LIN {X 0,Y 300.85,Z 546.983,A -85,B 0,C 180,E1 1983.68,E2 1983.68} C_VEL
LIN {X 0,Y 306.335,Z 523.084,A -85,B 0,C 180,E1 1983.212,E2 1983.212} C_VEL
LIN {X 0,Y 309.917,Z 499.874,A -85,B 0,C 180,E1 1982.824,E2 1982.824} C_VEL
LIN {X 0,Y 321.366,Z 402.053,A -85,B 0,C 180,E1 1981.248,E2 1981.248} C_VEL
LIN {X 0,Y 320.937,Z 400.568,A -85,B 0,C 180,E1 1978.393,E2 1978.393} C_VEL
LIN {X 0,Y 321.124,Z 402.876,A -85,B 0,C 180,E1 1974.448,E2 1974.448} C_VEL
LIN {X 0,Y 307.919,Z 513.947,A -85,B 0,C 180,E1 1972.759,E2 1972.759} C_VEL
LIN {X 0,Y 303.476,Z 536.476,A -85,B 0,C 180,E1 1972.375,E2 1972.375} C_VEL
LIN {X 0,Y 297.372,Z 559.018,A -85,B 0,C 180,E1 1971.893,E2 1971.893} C_VEL
LIN {X 0,Y 290.292,Z 579.356,A -85,B 0,C 180,E1 1971.299,E2 1971.299} C_VEL
LIN {X 0,Y 281.315,Z 600.354,A -85,B 0,C 180,E1 1970.495,E2 1970.495} C_VEL
LIN {X 0,Y 271.469,Z 619.823,A -85,B 0,C 180,E1 1969.536,E2 1969.536} C_VEL
LIN {X 0,Y 260.309,Z 638.411,A -85,B 0,C 180,E1 1968.361,E2 1968.361} C_VEL
LIN {X 0,Y 247.458,Z 657.08,A -85,B 0,C 180,E1 1966.84,E2 1966.84} C_VEL
LIN {X 0,Y 234.799,Z 673.136,A -85,B 0,C 180,E1 1965.155,E2 1965.155} C_VEL
LIN {X 0,Y 220.615,Z 688.99,A -85,B 0,C 180,E1 1962.99,E2 1962.99} C_VEL
LIN {X 0,Y 205.942,Z 703.636,A -85,B 0,C 180,E1 1960.365,E2 1960.365} C_VEL
LIN {X 0,Y 190.94,Z 716.802,A -85,B 0,C 180,E1 1957.161,E2 1957.161} C_VEL
LIN {X 0,Y 175.091,Z 729.345,A -85,B 0,C 180,E1 1952.976,E2 1952.976} C_VEL
LIN {X 0,Y 160.324,Z 739.898,A -85,B 0,C 180,E1 1948.01,E2 1948.01} C_VEL
LIN {X 0,Y 146.292,Z 748.96,A -85,B 0,C 180,E1 1941.81,E2 1941.81} C_VEL
LIN {X 0,Y 133.673,Z 756.634,A -85,B 0,C 180,E1 1934.076,E2 1934.076} C_VEL
LIN {X 0,Y 123.681,Z 762.5,A -85,B 0,C 180,E1 1925.027,E2 1925.027} C_VEL
LIN {X 0,Y 116.775,Z 766.633,A -85,B 0,C 180,E1 1914.805,E2 1914.805} C_VEL
LIN {X 0,Y 113.23,Z 769.201,A -85,B 0,C 180,E1 1904.314,E2 1904.314} C_VEL
LIN {X 0,Y 112.174,Z 770.206,A -85,B 0,C 180,E1 1894.601,E2 1894.601} C_VEL
LIN {X 0,Y 112.127,Z 770.283,A -85,B 0,C 180,E1 1887.118,E2 1887.118} C_VEL
LIN {X 0,Y 112.706,Z 769.615,A -85,B 0,C 180,E1 1878.746,E2 1878.746} C_VEL
LIN {X 0,Y 115.591,Z 767.48,A -85,B 0,C 180,E1 1867.753,E2 1867.753} C_VEL
LIN {X 0,Y 121.421,Z 763.846,A -85,B 0,C 180,E1 1857.64,E2 1857.64} C_VEL
LIN {X 0,Y 131.081,Z 758.196,A -85,B 0,C 180,E1 1847.838,E2 1847.838} C_VEL
LIN {X 0,Y 143.143,Z 751.061,A -85,B 0,C 180,E1 1839.796,E2 1839.796} C_VEL
LIN {X 0,Y 157.037,Z 742.16,A -85,B 0,C 180,E1 1833.201,E2 1833.201} C_VEL
LIN {X 0,Y 171.955,Z 731.773,A -85,B 0,C 180,E1 1827.895,E2 1827.895} C_VEL
LIN {X 0,Y 186.811,Z 720.428,A -85,B 0,C 180,E1 1823.765,E2 1823.765} C_VEL
LIN {X 0,Y 201.625,Z 707.683,A -85,B 0,C 180,E1 1820.41,E2 1820.41} C_VEL
LIN {X 0,Y 217.043,Z 692.931,A -85,B 0,C 180,E1 1817.529,E2 1817.529} C_VEL
LIN {X 0,Y 231.146,Z 677.659,A -85,B 0,C 180,E1 1815.292,E2 1815.292} C_VEL
LIN {X 0,Y 245.108,Z 660.462,A -85,B 0,C 180,E1 1813.375,E2 1813.375} C_VEL
LIN {X 0,Y 257.937,Z 642.496,A -85,B 0,C 180,E1 1811.832,E2 1811.832} C_VEL
LIN {X 0,Y 269.068,Z 624.347,A -85,B 0,C 180,E1 1810.625,E2 1810.625} C_VEL
LIN {X 0,Y 280.314,Z 602.942,A -85,B 0,C 180,E1 1809.521,E2 1809.521} C_VEL
LIN {X 0,Y 289.288,Z 582.628,A -85,B 0,C 180,E1 1808.711,E2 1808.711} C_VEL
LIN {X 0,Y 296.888,Z 561.22,A -85,B 0,C 180,E1 1808.067,E2 1808.067} C_VEL
LIN {X 0,Y 303.507,Z 537.366,A -85,B 0,C 180,E1 1807.547,E2 1807.547} C_VEL
LIN {X 0,Y 308.067,Z 514.578,A -85,B 0,C 180,E1 1807.157,E2 1807.157} C_VEL
LIN {X 0,Y 318.488,Z 427.457,A -85,B 0,C 180,E1 1805.83,E2 1805.83} C_VEL
LIN {X 0,Y 321.368,Z 402.948,A -85,B 0,C 180,E1 1805.445,E2 1805.445} C_VEL
LIN {X 0,Y 321.176,Z 400.924,A -85,B 0,C 180,E1 1801.427,E2 1801.427} C_VEL
LIN {X 0,Y 321.579,Z 402.546,A -85,B 0,C 180,E1 1798.708,E2 1798.708} C_VEL
LIN {X 0,Y 308.318,Z 513.24,A -85,B 0,C 180,E1 1796.963,E2 1796.963} C_VEL
LIN {X 0,Y 305.949,Z 526.418,A -85,B 0,C 180,E1 1796.734,E2 1796.734} C_VEL
LIN {X 0,Y 304.314,Z 534.011,A -85,B 0,C 180,E1 1796.782,E2 1796.782} C_VEL
LIN {X 0,Y 298.825,Z 552.994,A -85,B 0,C 180,E1 1797.537,E2 1797.537} C_VEL
LIN {X 0,Y 296.424,Z 560.346,A -85,B 0,C 180,E1 1797.555,E2 1797.555} C_VEL
LIN {X 0,Y 288.862,Z 581.554,A -85,B 0,C 180,E1 1796.943,E2 1796.943} C_VEL
LIN {X 0,Y 280.061,Z 601.523,A -85,B 0,C 180,E1 1796.2,E2 1796.2} C_VEL
LIN {X 0,Y 269.874,Z 621.266,A -85,B 0,C 180,E1 1795.268,E2 1795.268} C_VEL
LIN {X 0,Y 258.314,Z 640.207,A -85,B 0,C 180,E1 1794.122,E2 1794.122} C_VEL
LIN {X 0,Y 244.7,Z 659.572,A -85,B 0,C 180,E1 1792.608,E2 1792.608} C_VEL
LIN {X 0,Y 230.893,Z 676.781,A -85,B 0,C 180,E1 1790.86,E2 1790.86} C_VEL
LIN {X 0,Y 215.849,Z 693.137,A -85,B 0,C 180,E1 1788.663,E2 1788.663} C_VEL
LIN {X 0,Y 199.979,Z 708.528,A -85,B 0,C 180,E1 1785.915,E2 1785.915} C_VEL
LIN {X 0,Y 184.365,Z 722.031,A -85,B 0,C 180,E1 1782.644,E2 1782.644} C_VEL
LIN {X 0,Y 167.831,Z 734.817,A -85,B 0,C 180,E1 1778.333,E2 1778.333} C_VEL
LIN {X 0,Y 152.166,Z 745.889,A -85,B 0,C 180,E1 1773.039,E2 1773.039} C_VEL
LIN {X 0,Y 137.685,Z 755.245,A -85,B 0,C 180,E1 1766.503,E2 1766.503} C_VEL
LIN {X 0,Y 124.167,Z 763.536,A -85,B 0,C 180,E1 1757.8,E2 1757.8} C_VEL
LIN {X 0,Y 114.104,Z 769.775,A -85,B 0,C 180,E1 1747.834,E2 1747.834} C_VEL
LIN {X 0,Y 107.643,Z 774.053,A -85,B 0,C 180,E1 1736.913,E2 1736.913} C_VEL
LIN {X 0,Y 104.582,Z 776.871,A -85,B 0,C 180,E1 1725.527,E2 1725.527} C_VEL
LIN {X 0,Y 104.042,Z 778.016,A -85,B 0,C 180,E1 1715.515,E2 1715.515} C_VEL
LIN {X 0,Y 104.082,Z 778.19,A -85,B 0,C 180,E1 1708.349,E2 1708.349} C_VEL
LIN {X 0,Y 104.104,Z 777.613,A -85,B 0,C 180,E1 1700.045,E2 1700.045} C_VEL
LIN {X 0,Y 105.275,Z 776.015,A -85,B 0,C 180,E1 1690.585,E2 1690.585} C_VEL
LIN {X 0,Y 109.559,Z 772.724,A -85,B 0,C 180,E1 1679.076,E2 1679.076} C_VEL
LIN {X 0,Y 117.382,Z 767.616,A -85,B 0,C 180,E1 1668.365,E2 1668.365} C_VEL
LIN {X 0,Y 128.576,Z 760.822,A -85,B 0,C 180,E1 1658.957,E2 1658.957} C_VEL
LIN {X 0,Y 141.779,Z 752.578,A -85,B 0,C 180,E1 1651.428,E2 1651.428} C_VEL
LIN {X 0,Y 156.899,Z 742.51,A -85,B 0,C 180,E1 1645.192,E2 1645.192} C_VEL
LIN {X 0,Y 172.685,Z 731.153,A -85,B 0,C 180,E1 1640.288,E2 1640.288} C_VEL
LIN {X 0,Y 188.628,Z 718.295,A -85,B 0,C 180,E1 1636.383,E2 1636.383} C_VEL
LIN {X 0,Y 205.301,Z 703.363,A -85,B 0,C 180,E1 1633.09,E2 1633.09} C_VEL
LIN {X 0,Y 220.713,Z 687.911,A -85,B 0,C 180,E1 1630.577,E2 1630.577} C_VEL
LIN {X 0,Y 235.174,Z 671.347,A -85,B 0,C 180,E1 1628.557,E2 1628.557} C_VEL
LIN {X 0,Y 249.238,Z 653.14,A -85,B 0,C 180,E1 1626.852,E2 1626.852} C_VEL
LIN {X 0,Y 261.669,Z 634.646,A -85,B 0,C 180,E1 1625.518,E2 1625.518} C_VEL
LIN {X 0,Y 273.256,Z 614.539,A -85,B 0,C 180,E1 1624.393,E2 1624.393} C_VEL
LIN {X 0,Y 282.991,Z 594.865,A -85,B 0,C 180,E1 1623.536,E2 1623.536} C_VEL
LIN {X 0,Y 291.31,Z 574.448,A -85,B 0,C 180,E1 1622.845,E2 1622.845} C_VEL
LIN {X 0,Y 298.806,Z 551.771,A -85,B 0,C 180,E1 1622.256,E2 1622.256} C_VEL
LIN {X 0,Y 304.384,Z 529.797,A -85,B 0,C 180,E1 1621.828,E2 1621.828} C_VEL
LIN {X 0,Y 308.359,Z 506.904,A -85,B 0,C 180,E1 1621.453,E2 1621.453} C_VEL
LIN {X 0,Y 320.097,Z 409.255,A -85,B 0,C 180,E1 1619.96,E2 1619.96} C_VEL
LIN {X 0,Y 319.937,Z 408.589,A -85,B 0,C 180,E1 1618.209,E2 1618.209} C_VEL
LIN {X 0,Y 319.912,Z 410.101,A -85,B 0,C 180,E1 1615.774,E2 1615.774} C_VEL
LIN {X 0,Y 307.308,Z 513.987,A -85,B 0,C 180,E1 1614.248,E2 1614.248} C_VEL
LIN {X 0,Y 302.797,Z 536.523,A -85,B 0,C 180,E1 1613.885,E2 1613.885} C_VEL
LIN {X 0,Y 296.587,Z 559.159,A -85,B 0,C 180,E1 1613.433,E2 1613.433} C_VEL
LIN {X 0,Y 289.674,Z 578.813,A -85,B 0,C 180,E1 1612.897,E2 1612.897} C_VEL
LIN {X 0,Y 280.584,Z 599.936,A -85,B 0,C 180,E1 1612.147,E2 1612.147} C_VEL
LIN {X 0,Y 270.603,Z 619.466,A -85,B 0,C 180,E1 1611.252,E2 1611.252} C_VEL
LIN {X 0,Y 259.277,Z 638.131,A -85,B 0,C 180,E1 1610.151,E2 1610.151} C_VEL
LIN {X 0,Y 246.212,Z 656.875,A -85,B 0,C 180,E1 1608.723,E2 1608.723} C_VEL
LIN {X 0,Y 232.859,Z 673.513,A -85,B 0,C 180,E1 1607.077,E2 1607.077} C_VEL
LIN {X 0,Y 218.38,Z 689.339,A -85,B 0,C 180,E1 1605.025,E2 1605.025} C_VEL
LIN {X 0,Y 203.355,Z 703.968,A -85,B 0,C 180,E1 1602.522,E2 1602.522} C_VEL
LIN {X 0,Y 187.821,Z 717.21,A -85,B 0,C 180,E1 1599.43,E2 1599.43} C_VEL
LIN {X 0,Y 170.734,Z 730.213,A -85,B 0,C 180,E1 1595.188,E2 1595.188} C_VEL
LIN {X 0,Y 155.403,Z 740.705,A -85,B 0,C 180,E1 1590.292,E2 1590.292} C_VEL
LIN {X 0,Y 140.71,Z 749.653,A -85,B 0,C 180,E1 1584.1,E2 1584.1} C_VEL
LIN {X 0,Y 126.808,Z 757.516,A -85,B 0,C 180,E1 1575.848,E2 1575.848} C_VEL
LIN {X 0,Y 116.248,Z 763.28,A -85,B 0,C 180,E1 1566.403,E2 1566.403} C_VEL
LIN {X 0,Y 108.918,Z 767.232,A -85,B 0,C 180,E1 1555.559,E2 1555.559} C_VEL
LIN {X 0,Y 105.094,Z 769.696,A -85,B 0,C 180,E1 1543.759,E2 1543.759} C_VEL
LIN {X 0,Y 104.17,Z 770.517,A -85,B 0,C 180,E1 1534.404,E2 1534.404} C_VEL
LIN {X 0,Y 104.138,Z 770.566,A -85,B 0,C 180,E1 1526.698,E2 1526.698} C_VEL
LIN {X 0,Y 104.809,Z 769.907,A -85,B 0,C 180,E1 1517.885,E2 1517.885} C_VEL
LIN {X 0,Y 107.958,Z 767.878,A -85,B 0,C 180,E1 1506.478,E2 1506.478} C_VEL
LIN {X 0,Y 114.601,Z 764.142,A -85,B 0,C 180,E1 1495.452,E2 1495.452} C_VEL
LIN {X 0,Y 125.128,Z 758.495,A -85,B 0,C 180,E1 1485.319,E2 1485.319} C_VEL
LIN {X 0,Y 138.038,Z 751.362,A -85,B 0,C 180,E1 1477.18,E2 1477.18} C_VEL
LIN {X 0,Y 152.396,Z 742.65,A -85,B 0,C 180,E1 1470.744,E2 1470.744} C_VEL
LIN {X 0,Y 168.282,Z 732.081,A -85,B 0,C 180,E1 1465.433,E2 1465.433} C_VEL
LIN {X 0,Y 184.051,Z 720.452,A -85,B 0,C 180,E1 1461.345,E2 1461.345} C_VEL
LIN {X 0,Y 199.798,Z 707.246,A -85,B 0,C 180,E1 1458.048,E2 1458.048} C_VEL
LIN {X 0,Y 216.522,Z 691.447,A -85,B 0,C 180,E1 1455.182,E2 1455.182} C_VEL
LIN {X 0,Y 231.427,Z 675.489,A -85,B 0,C 180,E1 1453.037,E2 1453.037} C_VEL
LIN {X 0,Y 244.759,Z 659.044,A -85,B 0,C 180,E1 1451.365,E2 1451.365} C_VEL
LIN {X 0,Y 258.284,Z 640.025,A -85,B 0,C 180,E1 1449.876,E2 1449.876} C_VEL
LIN {X 0,Y 269.648,Z 621.523,A -85,B 0,C 180,E1 1448.758,E2 1448.758} C_VEL
LIN {X 0,Y 280.105,Z 601.418,A -85,B 0,C 180,E1 1447.816,E2 1447.816} C_VEL
LIN {X 0,Y 289.148,Z 580.835,A -85,B 0,C 180,E1 1447.068,E2 1447.068} C_VEL
LIN {X 0,Y 296.509,Z 560.122,A -85,B 0,C 180,E1 1446.495,E2 1446.495} C_VEL
LIN {X 0,Y 302.967,Z 536.836,A -85,B 0,C 180,E1 1446.027,E2 1446.027} C_VEL
LIN {X 0,Y 307.541,Z 514.047,A -85,B 0,C 180,E1 1445.66,E2 1445.66} C_VEL
LIN {X 0,Y 320.161,Z 410.157,A -85,B 0,C 180,E1 1444.13,E2 1444.13} C_VEL
LIN {X 0,Y 320.213,Z 408.924,A -85,B 0,C 180,E1 1441.253,E2 1441.253} C_VEL
LIN {X 0,Y 320.313,Z 409.713,A -85,B 0,C 180,E1 1440.029,E2 1440.029} C_VEL
LIN {X 0,Y 307.67,Z 513.462,A -85,B 0,C 180,E1 1438.447,E2 1438.447} C_VEL
LIN {X 0,Y 303.121,Z 536.211,A -85,B 0,C 180,E1 1438.064,E2 1438.064} C_VEL
LIN {X 0,Y 296.906,Z 558.879,A -85,B 0,C 180,E1 1437.591,E2 1437.591} C_VEL
LIN {X 0,Y 296.424,Z 560.346,A -85,B 0,C 180,E1 1437.555,E2 1437.555} C_VEL
LIN {X 0,Y 293.85,Z 567.982,A -85,B 0,C 180,E1 1437.556,E2 1437.556} C_VEL
LIN {X 0,Y 286.355,Z 586.249,A -85,B 0,C 180,E1 1438.198,E2 1438.198} C_VEL
LIN {X 0,Y 283.288,Z 593.171,A -85,B 0,C 180,E1 1438.161,E2 1438.161} C_VEL
LIN {X 0,Y 273.245,Z 613.523,A -85,B 0,C 180,E1 1437.351,E2 1437.351} C_VEL
LIN {X 0,Y 261.986,Z 633.058,A -85,B 0,C 180,E1 1436.353,E2 1436.353} C_VEL
LIN {X 0,Y 249.36,Z 651.677,A -85,B 0,C 180,E1 1435.125,E2 1435.125} C_VEL
LIN {X 0,Y 234.477,Z 670.763,A -85,B 0,C 180,E1 1433.48,E2 1433.48} C_VEL
LIN {X 0,Y 220.038,Z 687.044,A -85,B 0,C 180,E1 1431.639,E2 1431.639} C_VEL
LIN {X 0,Y 204.107,Z 702.714,A -85,B 0,C 180,E1 1429.272,E2 1429.272} C_VEL
LIN {X 0,Y 186.446,Z 718.124,A -85,B 0,C 180,E1 1426.078,E2 1426.078} C_VEL
LIN {X 0,Y 169.965,Z 730.956,A -85,B 0,C 180,E1 1422.359,E2 1422.359} C_VEL
LIN {X 0,Y 153.519,Z 742.298,A -85,B 0,C 180,E1 1417.64,E2 1417.64} C_VEL
LIN {X 0,Y 136.614,Z 752.921,A -85,B 0,C 180,E1 1411.116,E2 1411.116} C_VEL
LIN {X 0,Y 122.252,Z 761.316,A -85,B 0,C 180,E1 1403.272,E2 1403.272} C_VEL
LIN {X 0,Y 110.321,Z 767.897,A -85,B 0,C 180,E1 1393.528,E2 1393.528} C_VEL
LIN {X 0,Y 101.518,Z 773.023,A -85,B 0,C 180,E1 1381.466,E2 1381.466} C_VEL
LIN {X 0,Y 97.303,Z 775.984,A -85,B 0,C 180,E1 1369.821,E2 1369.821} C_VEL
LIN {X 0,Y 96.071,Z 777.613,A -85,B 0,C 180,E1 1358.378,E2 1358.378} C_VEL
LIN {X 0,Y 96.107,Z 777.966,A -85,B 0,C 180,E1 1350,E2 1350} C_VEL
LIN {X 0,Y 96.073,Z 777.583,A -85,B 0,C 180,E1 1341.368,E2 1341.368} C_VEL
LIN {X 0,Y 97.438,Z 775.84,A -85,B 0,C 180,E1 1329.581,E2 1329.581} C_VEL
LIN {X 0,Y 101.817,Z 772.822,A -85,B 0,C 180,E1 1317.976,E2 1317.976} C_VEL
LIN {X 0,Y 110.324,Z 767.845,A -85,B 0,C 180,E1 1306.468,E2 1306.468} C_VEL
LIN {X 0,Y 122.247,Z 761.249,A -85,B 0,C 180,E1 1296.725,E2 1296.725} C_VEL
LIN {X 0,Y 136.592,Z 752.85,A -85,B 0,C 180,E1 1288.889,E2 1288.889} C_VEL
LIN {X 0,Y 152.72,Z 742.723,A -85,B 0,C 180,E1 1282.617,E2 1282.617} C_VEL
LIN {X 0,Y 169.112,Z 731.441,A -85,B 0,C 180,E1 1277.849,E2 1277.849} C_VEL
LIN {X 0,Y 185.555,Z 718.683,A -85,B 0,C 180,E1 1274.094,E2 1274.094} C_VEL
LIN {X 0,Y 202.659,Z 703.879,A -85,B 0,C 180,E1 1270.955,E2 1270.955} C_VEL
LIN {X 0,Y 217.935,Z 688.97,A -85,B 0,C 180,E1 1268.637,E2 1268.637} C_VEL
LIN {X 0,Y 232.566,Z 672.763,A -85,B 0,C 180,E1 1266.736,E2 1266.736} C_VEL
LIN {X 0,Y 246.46,Z 655.418,A -85,B 0,C 180,E1 1265.169,E2 1265.169} C_VEL
LIN {X 0,Y 259.544,Z 636.425,A -85,B 0,C 180,E1 1263.858,E2 1263.858} C_VEL
LIN {X 0,Y 271.77,Z 615.824,A -85,B 0,C 180,E1 1262.762,E2 1262.762} C_VEL
LIN {X 0,Y 282.111,Z 595.339,A -85,B 0,C 180,E1 1261.922,E2 1261.922} C_VEL
LIN {X 0,Y 290.523,Z 574.999,A -85,B 0,C 180,E1 1261.28,E2 1261.28} C_VEL
LIN {X 0,Y 298.052,Z 552.671,A -85,B 0,C 180,E1 1260.736,E2 1260.736} C_VEL
LIN {X 0,Y 303.637,Z 531.077,A -85,B 0,C 180,E1 1260.34,E2 1260.34} C_VEL
LIN {X 0,Y 307.8,Z 507.983,A -85,B 0,C 180,E1 1259.98,E2 1259.98} C_VEL
LIN {X 0,Y 318.99,Z 416.494,A -85,B 0,C 180,E1 1258.608,E2 1258.608} C_VEL
LIN {X 0,Y 318.871,Z 417.333,A -85,B 0,C 180,E1 1257.109,E2 1257.109} C_VEL
LIN {X 0,Y 306.904,Z 514.026,A -85,B 0,C 180,E1 1255.742,E2 1255.742} C_VEL
LIN {X 0,Y 302.298,Z 536.708,A -85,B 0,C 180,E1 1255.398,E2 1255.398} C_VEL
LIN {X 0,Y 296.084,Z 559.1,A -85,B 0,C 180,E1 1254.983,E2 1254.983} C_VEL
LIN {X 0,Y 288.797,Z 579.545,A -85,B 0,C 180,E1 1254.466,E2 1254.466} C_VEL
LIN {X 0,Y 279.605,Z 600.515,A -85,B 0,C 180,E1 1253.769,E2 1253.769} C_VEL
LIN {X 0,Y 269.501,Z 619.982,A -85,B 0,C 180,E1 1252.935,E2 1252.935} C_VEL
LIN {X 0,Y 258.025,Z 638.579,A -85,B 0,C 180,E1 1251.91,E2 1251.91} C_VEL
LIN {X 0,Y 245.071,Z 656.875,A -85,B 0,C 180,E1 1250.607,E2 1250.607} C_VEL
LIN {X 0,Y 231.65,Z 673.342,A -85,B 0,C 180,E1 1249.087,E2 1249.087} C_VEL
LIN {X 0,Y 216.427,Z 689.686,A -85,B 0,C 180,E1 1247.099,E2 1247.099} C_VEL
LIN {X 0,Y 200.899,Z 704.438,A -85,B 0,C 180,E1 1244.705,E2 1244.705} C_VEL
LIN {X 0,Y 184.627,Z 717.92,A -85,B 0,C 180,E1 1241.693,E2 1241.693} C_VEL
LIN {X 0,Y 167.467,Z 730.525,A -85,B 0,C 180,E1 1237.728,E2 1237.728} C_VEL
LIN {X 0,Y 151.512,Z 741.011,A -85,B 0,C 180,E1 1232.983,E2 1232.983} C_VEL
LIN {X 0,Y 136.065,Z 749.956,A -85,B 0,C 180,E1 1226.897,E2 1226.897} C_VEL
LIN {X 0,Y 121.242,Z 757.813,A -85,B 0,C 180,E1 1218.628,E2 1218.628} C_VEL
LIN {X 0,Y 109.774,Z 763.578,A -85,B 0,C 180,E1 1208.936,E2 1208.936} C_VEL
LIN {X 0,Y 101.637,Z 767.528,A -85,B 0,C 180,E1 1197.539,E2 1197.539} C_VEL
LIN {X 0,Y 97.269,Z 769.99,A -85,B 0,C 180,E1 1184.891,E2 1184.891} C_VEL
LIN {X 0,Y 96.187,Z 770.808,A -85,B 0,C 180,E1 1174.77,E2 1174.77} C_VEL
LIN {X 0,Y 96.143,Z 770.868,A -85,B 0,C 180,E1 1166.748,E2 1166.748} C_VEL
LIN {X 0,Y 96.85,Z 770.262,A -85,B 0,C 180,E1 1157.479,E2 1157.479} C_VEL
LIN {X 0,Y 100.385,Z 768.276,A -85,B 0,C 180,E1 1145.012,E2 1145.012} C_VEL
LIN {X 0,Y 107.55,Z 764.636,A -85,B 0,C 180,E1 1133.489,E2 1133.489} C_VEL
LIN {X 0,Y 119.44,Z 758.793,A -85,B 0,C 180,E1 1122.554,E2 1122.554} C_VEL
LIN {X 0,Y 133.243,Z 751.663,A -85,B 0,C 180,E1 1114.369,E2 1114.369} C_VEL
LIN {X 0,Y 148.374,Z 742.949,A -85,B 0,C 180,E1 1108.024,E2 1108.024} C_VEL
LIN {X 0,Y 165.224,Z 732.188,A -85,B 0,C 180,E1 1102.787,E2 1102.787} C_VEL
LIN {X 0,Y 181.707,Z 720.409,A -85,B 0,C 180,E1 1098.841,E2 1098.841} C_VEL
LIN {X 0,Y 197.428,Z 707.566,A -85,B 0,C 180,E1 1095.802,E2 1095.802} C_VEL
LIN {X 0,Y 213.629,Z 692.698,A -85,B 0,C 180,E1 1093.224,E2 1093.224} C_VEL
LIN {X 0,Y 228.343,Z 677.36,A -85,B 0,C 180,E1 1091.242,E2 1091.242} C_VEL
LIN {X 0,Y 242.357,Z 660.631,A -85,B 0,C 180,E1 1089.605,E2 1089.605} C_VEL
LIN {X 0,Y 255.602,Z 642.645,A -85,B 0,C 180,E1 1088.25,E2 1088.25} C_VEL
LIN {X 0,Y 267.057,Z 624.485,A -85,B 0,C 180,E1 1087.194,E2 1087.194} C_VEL
LIN {X 0,Y 278.6,Z 603.078,A -85,B 0,C 180,E1 1086.233,E2 1086.233} C_VEL
LIN {X 0,Y 287.791,Z 582.774,A -85,B 0,C 180,E1 1085.531,E2 1085.531} C_VEL
LIN {X 0,Y 295.563,Z 561.409,A -85,B 0,C 180,E1 1084.973,E2 1084.973} C_VEL
LIN {X 0,Y 302.298,Z 537.76,A -85,B 0,C 180,E1 1084.526,E2 1084.526} C_VEL
LIN {X 0,Y 307.014,Z 514.966,A -85,B 0,C 180,E1 1084.18,E2 1084.18} C_VEL
LIN {X 0,Y 315.968,Z 443.369,A -85,B 0,C 180,E1 1083.167,E2 1083.167} C_VEL
LIN {X 0,Y 319.122,Z 417.372,A -85,B 0,C 180,E1 1082.784,E2 1082.784} C_VEL
LIN {X 0,Y 319.209,Z 416.958,A -85,B 0,C 180,E1 1081.36,E2 1081.36} C_VEL
LIN {X 0,Y 307.229,Z 513.683,A -85,B 0,C 180,E1 1079.937,E2 1079.937} C_VEL
LIN {X 0,Y 302.613,Z 536.45,A -85,B 0,C 180,E1 1079.576,E2 1079.576} C_VEL
LIN {X 0,Y 296.234,Z 559.362,A -85,B 0,C 180,E1 1079.129,E2 1079.129} C_VEL
LIN {X 0,Y 289.038,Z 579.526,A -85,B 0,C 180,E1 1078.596,E2 1078.596} C_VEL
LIN {X 0,Y 283.288,Z 593.171,A -85,B 0,C 180,E1 1078.161,E2 1078.161} C_VEL
LIN {X 0,Y 280.03,Z 600.219,A -85,B 0,C 180,E1 1078.108,E2 1078.108} C_VEL
LIN {X 0,Y 270.502,Z 617.76,A -85,B 0,C 180,E1 1078.649,E2 1078.649} C_VEL
LIN {X 0,Y 266.551,Z 624.394,A -85,B 0,C 180,E1 1078.554,E2 1078.554} C_VEL
LIN {X 0,Y 254.41,Z 643.457,A -85,B 0,C 180,E1 1077.523,E2 1077.523} C_VEL
LIN {X 0,Y 240.974,Z 661.506,A -85,B 0,C 180,E1 1076.254,E2 1076.254} C_VEL
LIN {X 0,Y 225.953,Z 679.199,A -85,B 0,C 180,E1 1074.63,E2 1074.63} C_VEL
LIN {X 0,Y 210.668,Z 694.954,A -85,B 0,C 180,E1 1072.709,E2 1072.709} C_VEL
LIN {X 0,Y 193.863,Z 710.172,A -85,B 0,C 180,E1 1070.201,E2 1070.201} C_VEL
LIN {X 0,Y 177.381,Z 723.486,A -85,B 0,C 180,E1 1067.196,E2 1067.196} C_VEL
LIN {X 0,Y 160.374,Z 735.563,A -85,B 0,C 180,E1 1063.335,E2 1063.335} C_VEL
LIN {X 0,Y 142.379,Z 747.005,A -85,B 0,C 180,E1 1057.964,E2 1057.964} C_VEL
LIN {X 0,Y 126.383,Z 756.231,A -85,B 0,C 180,E1 1051.418,E2 1051.418} C_VEL
LIN {X 0,Y 111.749,Z 763.877,A -85,B 0,C 180,E1 1042.778,E2 1042.778} C_VEL
LIN {X 0,Y 99.615,Z 770.049,A -85,B 0,C 180,E1 1031.486,E2 1031.486} C_VEL
LIN {X 0,Y 92.155,Z 774.09,A -85,B 0,C 180,E1 1019.224,E2 1019.224} C_VEL
LIN {X 0,Y 88.563,Z 776.584,A -85,B 0,C 180,E1 1005.721,E2 1005.721} C_VEL
LIN {X 0,Y 88.052,Z 777.458,A -85,B 0,C 180,E1 995.866,E2 995.866} C_VEL
LIN {X 0,Y 88.086,Z 777.608,A -85,B 0,C 180,E1 988.049,E2 988.049} C_VEL
LIN {X 0,Y 88.156,Z 777.098,A -85,B 0,C 180,E1 978.883,E2 978.883} C_VEL
LIN {X 0,Y 89.965,Z 775.418,A -85,B 0,C 180,E1 967.109,E2 967.109} C_VEL
LIN {X 0,Y 95.587,Z 772.178,A -85,B 0,C 180,E1 954.144,E2 954.144} C_VEL
LIN {X 0,Y 105.534,Z 766.979,A -85,B 0,C 180,E1 942.273,E2 942.273} C_VEL
LIN {X 0,Y 119.414,Z 759.837,A -85,B 0,C 180,E1 932.258,E2 932.258} C_VEL
LIN {X 0,Y 134.548,Z 751.54,A -85,B 0,C 180,E1 924.962,E2 924.962} C_VEL
LIN {X 0,Y 151.351,Z 741.345,A -85,B 0,C 180,E1 919.15,E2 919.15} C_VEL
LIN {X 0,Y 168.484,Z 729.852,A -85,B 0,C 180,E1 914.696,E2 914.696} C_VEL
LIN {X 0,Y 185.519,Z 716.924,A -85,B 0,C 180,E1 911.227,E2 911.227} C_VEL
LIN {X 0,Y 202.179,Z 702.674,A -85,B 0,C 180,E1 908.486,E2 908.486} C_VEL
LIN {X 0,Y 218.277,Z 687.196,A -85,B 0,C 180,E1 906.29,E2 906.29} C_VEL
LIN {X 0,Y 233.296,Z 670.57,A -85,B 0,C 180,E1 904.536,E2 904.536} C_VEL
LIN {X 0,Y 248.542,Z 651.277,A -85,B 0,C 180,E1 902.997,E2 902.997} C_VEL
LIN {X 0,Y 261.591,Z 632.222,A -85,B 0,C 180,E1 901.841,E2 901.841} C_VEL
LIN {X 0,Y 272.989,Z 612.554,A -85,B 0,C 180,E1 900.921,E2 900.921} C_VEL
LIN {X 0,Y 283.453,Z 591.256,A -85,B 0,C 180,E1 900.152,E2 900.152} C_VEL
LIN {X 0,Y 292.211,Z 569.689,A -85,B 0,C 180,E1 899.555,E2 899.555} C_VEL
LIN {X 0,Y 299.079,Z 548.087,A -85,B 0,C 180,E1 899.109,E2 899.109} C_VEL
LIN {X 0,Y 304.742,Z 524.632,A -85,B 0,C 180,E1 898.73,E2 898.73} C_VEL
LIN {X 0,Y 308.506,Z 501.749,A -85,B 0,C 180,E1 898.397,E2 898.397} C_VEL
LIN {X 0,Y 312.819,Z 466.535,A -85,B 0,C 180,E1 897.885,E2 897.885} C_VEL
LIN {X 0,Y 306.465,Z 515.586,A -85,B 0,C 180,E1 897.218,E2 897.218} C_VEL
LIN {X 0,Y 301.673,Z 538.312,A -85,B 0,C 180,E1 896.895,E2 896.895} C_VEL
LIN {X 0,Y 295.003,Z 561.412,A -85,B 0,C 180,E1 896.491,E2 896.491} C_VEL
LIN {X 0,Y 287.159,Z 582.778,A -85,B 0,C 180,E1 895.977,E2 895.977} C_VEL
LIN {X 0,Y 277.875,Z 603.085,A -85,B 0,C 180,E1 895.331,E2 895.331} C_VEL
LIN {X 0,Y 266.691,Z 623.692,A -85,B 0,C 180,E1 894.481,E2 894.481} C_VEL
LIN {X 0,Y 255.09,Z 641.932,A -85,B 0,C 180,E1 893.512,E2 893.512} C_VEL
LIN {X 0,Y 241.663,Z 660.068,A -85,B 0,C 180,E1 892.257,E2 892.257} C_VEL
LIN {X 0,Y 227.425,Z 676.917,A -85,B 0,C 180,E1 890.741,E2 890.741} C_VEL
LIN {X 0,Y 212.902,Z 691.858,A -85,B 0,C 180,E1 888.964,E2 888.964} C_VEL
LIN {X 0,Y 195.428,Z 707.66,A -85,B 0,C 180,E1 886.424,E2 886.424} C_VEL
LIN {X 0,Y 179.3,Z 720.519,A -85,B 0,C 180,E1 883.561,E2 883.561} C_VEL
LIN {X 0,Y 162.335,Z 732.297,A -85,B 0,C 180,E1 879.823,E2 879.823} C_VEL
LIN {X 0,Y 144.775,Z 743.107,A -85,B 0,C 180,E1 874.783,E2 874.783} C_VEL
LIN {X 0,Y 128.861,Z 751.835,A -85,B 0,C 180,E1 868.593,E2 868.593} C_VEL
LIN {X 0,Y 114.12,Z 758.99,A -85,B 0,C 180,E1 860.442,E2 860.442} C_VEL
LIN {X 0,Y 101.151,Z 764.862,A -85,B 0,C 180,E1 849.243,E2 849.243} C_VEL
LIN {X 0,Y 92.962,Z 768.595,A -85,B 0,C 180,E1 836.782,E2 836.782} C_VEL
LIN {X 0,Y 89.009,Z 770.532,A -85,B 0,C 180,E1 823.644,E2 823.644} C_VEL
LIN {X 0,Y 88.149,Z 771.161,A -85,B 0,C 180,E1 813.251,E2 813.251} C_VEL
LIN {X 0,Y 88.204,Z 771.107,A -85,B 0,C 180,E1 804.797,E2 804.797} C_VEL
LIN {X 0,Y 89.465,Z 770.307,A -85,B 0,C 180,E1 793.776,E2 793.776} C_VEL
LIN {X 0,Y 94.457,Z 767.878,A -85,B 0,C 180,E1 780.165,E2 780.165} C_VEL
LIN {X 0,Y 103.482,Z 763.945,A -85,B 0,C 180,E1 768.19,E2 768.19} C_VEL
LIN {X 0,Y 115.921,Z 758.214,A -85,B 0,C 180,E1 758.29,E2 758.29} C_VEL
LIN {X 0,Y 131.696,Z 750.392,A -85,B 0,C 180,E1 750.062,E2 750.062} C_VEL
LIN {X 0,Y 147.902,Z 741.457,A -85,B 0,C 180,E1 744.131,E2 744.131} C_VEL
LIN {X 0,Y 164.804,Z 730.792,A -85,B 0,C 180,E1 739.493,E2 739.493} C_VEL
LIN {X 0,Y 182.78,Z 717.975,A -85,B 0,C 180,E1 735.69,E2 735.69} C_VEL
LIN {X 0,Y 199.02,Z 704.853,A -85,B 0,C 180,E1 732.939,E2 732.939} C_VEL
LIN {X 0,Y 214.711,Z 690.298,A -85,B 0,C 180,E1 730.72,E2 730.72} C_VEL
LIN {X 0,Y 230.22,Z 674.027,A -85,B 0,C 180,E1 728.864,E2 728.864} C_VEL
LIN {X 0,Y 244.01,Z 657.41,A -85,B 0,C 180,E1 727.434,E2 727.434} C_VEL
LIN {X 0,Y 257.464,Z 638.72,A -85,B 0,C 180,E1 726.203,E2 726.203} C_VEL
LIN {X 0,Y 269.086,Z 620.122,A -85,B 0,C 180,E1 725.257,E2 725.257} C_VEL
LIN {X 0,Y 279.31,Z 600.657,A -85,B 0,C 180,E1 724.489,E2 724.489} C_VEL
LIN {X 0,Y 288.602,Z 579.719,A -85,B 0,C 180,E1 723.85,E2 723.85} C_VEL
LIN {X 0,Y 295.963,Z 559.299,A -85,B 0,C 180,E1 723.375,E2 723.375} C_VEL
LIN {X 0,Y 302.36,Z 536.489,A -85,B 0,C 180,E1 722.988,E2 722.988} C_VEL
LIN {X 0,Y 307.014,Z 513.722,A -85,B 0,C 180,E1 722.666,E2 722.666} C_VEL
LIN {X 0,Y 312.684,Z 469.731,A -85,B 0,C 180,E1 722.06,E2 722.06} C_VEL
LIN {X 0,Y 306.728,Z 515.57,A -85,B 0,C 180,E1 721.406,E2 721.406} C_VEL
LIN {X 0,Y 301.938,Z 538.268,A -85,B 0,C 180,E1 721.066,E2 721.066} C_VEL
LIN {X 0,Y 295.306,Z 561.246,A -85,B 0,C 180,E1 720.643,E2 720.643} C_VEL
LIN {X 0,Y 287.452,Z 582.663,A -85,B 0,C 180,E1 720.107,E2 720.107} C_VEL
LIN {X 0,Y 278.482,Z 602.35,A -85,B 0,C 180,E1 719.473,E2 719.473} C_VEL
LIN {X 0,Y 267.531,Z 622.769,A -85,B 0,C 180,E1 718.632,E2 718.632} C_VEL
LIN {X 0,Y 266.551,Z 624.394,A -85,B 0,C 180,E1 718.554,E2 718.554} C_VEL
LIN {X 0,Y 262.431,Z 631.157,A -85,B 0,C 180,E1 718.44,E2 718.44} C_VEL
LIN {X 0,Y 251.006,Z 647.521,A -85,B 0,C 180,E1 718.884,E2 718.884} C_VEL
LIN {X 0,Y 246.454,Z 653.632,A -85,B 0,C 180,E1 718.735,E2 718.735} C_VEL
LIN {X 0,Y 231.704,Z 671.703,A -85,B 0,C 180,E1 717.375,E2 717.375} C_VEL
LIN {X 0,Y 216.069,Z 688.483,A -85,B 0,C 180,E1 715.709,E2 715.709} C_VEL
LIN {X 0,Y 199.867,Z 703.661,A -85,B 0,C 180,E1 713.682,E2 713.682} C_VEL
LIN {X 0,Y 182.209,Z 718.188,A -85,B 0,C 180,E1 711.007,E2 711.007} C_VEL
LIN {X 0,Y 164.75,Z 730.931,A -85,B 0,C 180,E1 707.708,E2 707.708} C_VEL
LIN {X 0,Y 146.986,Z 742.264,A -85,B 0,C 180,E1 703.4,E2 703.4} C_VEL
LIN {X 0,Y 128.825,Z 752.578,A -85,B 0,C 180,E1 697.454,E2 697.454} C_VEL
LIN {X 0,Y 113.02,Z 760.704,A -85,B 0,C 180,E1 690.107,E2 690.107} C_VEL
LIN {X 0,Y 98.883,Z 767.289,A -85,B 0,C 180,E1 680.215,E2 680.215} C_VEL
LIN {X 0,Y 87.8,Z 772.423,A -85,B 0,C 180,E1 667.124,E2 667.124} C_VEL
LIN {X 0,Y 82.058,Z 775.389,A -85,B 0,C 180,E1 653.709,E2 653.709} C_VEL
LIN {X 0,Y 80.094,Z 777.048,A -85,B 0,C 180,E1 639.536,E2 639.536} C_VEL
LIN {X 0,Y 80.116,Z 777.384,A -85,B 0,C 180,E1 630,E2 630} C_VEL
LIN {X 0,Y 80.096,Z 777.043,A -85,B 0,C 180,E1 620.458,E2 620.458} C_VEL
LIN {X 0,Y 82.058,Z 775.365,A -85,B 0,C 180,E1 606.291,E2 606.291} C_VEL
LIN {X 0,Y 87.823,Z 772.38,A -85,B 0,C 180,E1 592.837,E2 592.837} C_VEL
LIN {X 0,Y 98.881,Z 767.236,A -85,B 0,C 180,E1 579.783,E2 579.783} C_VEL
LIN {X 0,Y 113.016,Z 760.63,A -85,B 0,C 180,E1 569.89,E2 569.89} C_VEL
LIN {X 0,Y 128.821,Z 752.487,A -85,B 0,C 180,E1 562.541,E2 562.541} C_VEL
LIN {X 0,Y 147.081,Z 742.09,A -85,B 0,C 180,E1 556.566,E2 556.566} C_VEL
LIN {X 0,Y 164.905,Z 730.7,A -85,B 0,C 180,E1 552.252,E2 552.252} C_VEL
LIN {X 0,Y 182.205,Z 718.029,A -85,B 0,C 180,E1 548.984,E2 548.984} C_VEL
LIN {X 0,Y 200.163,Z 703.193,A -85,B 0,C 180,E1 546.268,E2 546.268} C_VEL
LIN {X 0,Y 216.552,Z 687.792,A -85,B 0,C 180,E1 544.226,E2 544.226} C_VEL
LIN {X 0,Y 231.702,Z 671.433,A -85,B 0,C 180,E1 542.613,E2 542.613} C_VEL
LIN {X 0,Y 246.516,Z 653.209,A -85,B 0,C 180,E1 541.247,E2 541.247} C_VEL
LIN {X 0,Y 259.457,Z 634.769,A -85,B 0,C 180,E1 540.192,E2 540.192} C_VEL
LIN {X 0,Y 271.474,Z 614.751,A -85,B 0,C 180,E1 539.308,E2 539.308} C_VEL
LIN {X 0,Y 281.532,Z 595.167,A -85,B 0,C 180,E1 538.637,E2 538.637} C_VEL
LIN {X 0,Y 290.11,Z 574.799,A -85,B 0,C 180,E1 538.098,E2 538.098} C_VEL
LIN {X 0,Y 292.715,Z 567.909,A -85,B 0,C 180,E1 537.925,E2 537.925} C_VEL
LIN {X 0,Y 284.239,Z 589.029,A -85,B 0,C 180,E1 537.423,E2 537.423} C_VEL
LIN {X 0,Y 274.386,Z 609.457,A -85,B 0,C 180,E1 536.781,E2 536.781} C_VEL
LIN {X 0,Y 263.59,Z 628.189,A -85,B 0,C 180,E1 536.023,E2 536.023} C_VEL
LIN {X 0,Y 250.411,Z 647.789,A -85,B 0,C 180,E1 534.998,E2 534.998} C_VEL
LIN {X 0,Y 236.844,Z 665.272,A -85,B 0,C 180,E1 533.802,E2 533.802} C_VEL
LIN {X 0,Y 221.958,Z 681.783,A -85,B 0,C 180,E1 532.312,E2 532.312} C_VEL
LIN {X 0,Y 205.836,Z 697.496,A -85,B 0,C 180,E1 530.42,E2 530.42} C_VEL
LIN {X 0,Y 189.053,Z 711.776,A -85,B 0,C 180,E1 528.068,E2 528.068} C_VEL
LIN {X 0,Y 171.752,Z 724.596,A -85,B 0,C 180,E1 525.093,E2 525.093} C_VEL
LIN {X 0,Y 154.149,Z 736.101,A -85,B 0,C 180,E1 521.258,E2 521.258} C_VEL
LIN {X 0,Y 137.382,Z 745.649,A -85,B 0,C 180,E1 516.49,E2 516.49} C_VEL
LIN {X 0,Y 120.29,Z 754.221,A -85,B 0,C 180,E1 509.818,E2 509.818} C_VEL
LIN {X 0,Y 105.22,Z 761.009,A -85,B 0,C 180,E1 501.186,E2 501.186} C_VEL
LIN {X 0,Y 92.995,Z 765.948,A -85,B 0,C 180,E1 490.172,E2 490.172} C_VEL
LIN {X 0,Y 84.333,Z 769.422,A -85,B 0,C 180,E1 476.019,E2 476.019} C_VEL
LIN {X 0,Y 80.863,Z 771.013,A -85,B 0,C 180,E1 462.86,E2 462.86} C_VEL
LIN {X 0,Y 80.132,Z 771.516,A -85,B 0,C 180,E1 451.43,E2 451.43} C_VEL
LIN {X 0,Y 80.456,Z 771.301,A -85,B 0,C 180,E1 440.703,E2 440.703} C_VEL
LIN {X 0,Y 83.534,Z 769.78,A -85,B 0,C 180,E1 425.986,E2 425.986} C_VEL
LIN {X 0,Y 91.116,Z 766.801,A -85,B 0,C 180,E1 412.085,E2 412.085} C_VEL
LIN {X 0,Y 102.696,Z 762.067,A -85,B 0,C 180,E1 400.589,E2 400.589} C_VEL
LIN {X 0,Y 118.382,Z 755.198,A -85,B 0,C 180,E1 391.012,E2 391.012} C_VEL
LIN {X 0,Y 134.897,Z 747.127,A -85,B 0,C 180,E1 384.266,E2 384.266} C_VEL
LIN {X 0,Y 152.367,Z 737.256,A -85,B 0,C 180,E1 379.104,E2 379.104} C_VEL
LIN {X 0,Y 170.801,Z 725.399,A -85,B 0,C 180,E1 375.012,E2 375.012} C_VEL
LIN {X 0,Y 188.081,Z 712.759,A -85,B 0,C 180,E1 372.004,E2 372.004} C_VEL
LIN {X 0,Y 204.849,Z 698.569,A -85,B 0,C 180,E1 369.625,E2 369.625} C_VEL
LIN {X 0,Y 221.441,Z 682.566,A -85,B 0,C 180,E1 367.665,E2 367.665} C_VEL
LIN {X 0,Y 236.328,Z 666.179,A -85,B 0,C 180,E1 366.167,E2 366.167} C_VEL
LIN {X 0,Y 249.896,Z 648.827,A -85,B 0,C 180,E1 364.968,E2 364.968} C_VEL
LIN {X 0,Y 263.077,Z 629.445,A -85,B 0,C 180,E1 363.938,E2 363.938} C_VEL
LIN {X 0,Y 273.874,Z 610.839,A -85,B 0,C 180,E1 363.176,E2 363.176} C_VEL
LIN {X 0,Y 284.222,Z 589.641,A -85,B 0,C 180,E1 362.501,E2 362.501} C_VEL
LIN {X 0,Y 292.289,Z 569.856,A -85,B 0,C 180,E1 362.021,E2 362.021} C_VEL
LIN {X 0,Y 283.547,Z 591.172,A -85,B 0,C 180,E1 361.484,E2 361.484} C_VEL
LIN {X 0,Y 272.979,Z 612.474,A -85,B 0,C 180,E1 360.783,E2 360.783} C_VEL
LIN {X 0,Y 261.456,Z 632.143,A -85,B 0,C 180,E1 359.943,E2 359.943} C_VEL
LIN {X 0,Y 248.503,Z 650.839,A -85,B 0,C 180,E1 358.91,E2 358.91} C_VEL
LIN {X 0,Y 246.454,Z 653.632,A -85,B 0,C 180,E1 358.735,E2 358.735} C_VEL
LIN {X 0,Y 241.723,Z 659.756,A -85,B 0,C 180,E1 358.564,E2 358.564} C_VEL
LIN {X 0,Y 228.455,Z 674.839,A -85,B 0,C 180,E1 358.893,E2 358.893} C_VEL
LIN {X 0,Y 223.152,Z 680.407,A -85,B 0,C 180,E1 358.66,E2 358.66} C_VEL
LIN {X 0,Y 206.712,Z 696.634,A -85,B 0,C 180,E1 356.95,E2 356.95} C_VEL
LIN {X 0,Y 189.732,Z 711.137,A -85,B 0,C 180,E1 354.855,E2 354.855} C_VEL
LIN {X 0,Y 170.516,Z 725.549,A -85,B 0,C 180,E1 351.91,E2 351.91} C_VEL
LIN {X 0,Y 152.13,Z 737.655,A -85,B 0,C 180,E1 348.31,E2 348.31} C_VEL
LIN {X 0,Y 134.355,Z 747.805,A -85,B 0,C 180,E1 343.736,E2 343.736} C_VEL
LIN {X 0,Y 115.262,Z 757.466,A -85,B 0,C 180,E1 336.852,E2 336.852} C_VEL
LIN {X 0,Y 99.004,Z 764.841,A -85,B 0,C 180,E1 328.028,E2 328.028} C_VEL
LIN {X 0,Y 85.666,Z 770.322,A -85,B 0,C 180,E1 316.354,E2 316.354} C_VEL
LIN {X 0,Y 76.178,Z 774.349,A -85,B 0,C 180,E1 300.789,E2 300.789} C_VEL
LIN {X 0,Y 72.638,Z 776.22,A -85,B 0,C 180,E1 286.802,E2 286.802} C_VEL
LIN {X 0,Y 72.06,Z 776.954,A -85,B 0,C 180,E1 274.775,E2 274.775} C_VEL
LIN {X 0,Y 72.076,Z 777.001,A -85,B 0,C 180,E1 266.819,E2 266.819} C_VEL
LIN {X 0,Y 72.427,Z 776.384,A -85,B 0,C 180,E1 255.089,E2 255.089} C_VEL
LIN {X 0,Y 75.611,Z 774.573,A -85,B 0,C 180,E1 240.708,E2 240.708} C_VEL
LIN {X 0,Y 84.64,Z 770.714,A -85,B 0,C 180,E1 224.866,E2 224.866} C_VEL
LIN {X 0,Y 96.984,Z 765.594,A -85,B 0,C 180,E1 213.38,E2 213.38} C_VEL
LIN {X 0,Y 112.907,Z 758.482,A -85,B 0,C 180,E1 204.202,E2 204.202} C_VEL
LIN {X 0,Y 130.063,Z 750.069,A -85,B 0,C 180,E1 197.594,E2 197.594} C_VEL
LIN {X 0,Y 148.5,Z 739.661,A -85,B 0,C 180,E1 192.508,E2 192.508} C_VEL
LIN {X 0,Y 167.836,Z 727.255,A -85,B 0,C 180,E1 188.548,E2 188.548} C_VEL
LIN {X 0,Y 185.881,Z 714.094,A -85,B 0,C 180,E1 185.678,E2 185.678} C_VEL
LIN {X 0,Y 203.329,Z 699.407,A -85,B 0,C 180,E1 183.427,E2 183.427} C_VEL
LIN {X 0,Y 220.808,Z 682.592,A -85,B 0,C 180,E1 181.556,E2 181.556} C_VEL
LIN {X 0,Y 235.961,Z 665.955,A -85,B 0,C 180,E1 180.186,E2 180.186} C_VEL
LIN {X 0,Y 249.99,Z 648.045,A -85,B 0,C 180,E1 179.069,E2 179.069} C_VEL
LIN {X 0,Y 263.598,Z 627.954,A -85,B 0,C 180,E1 178.112,E2 178.112} C_VEL
LIN {X 0,Y 265.936,Z 624.156,A -85,B 0,C 180,E1 177.943,E2 177.943} C_VEL
LIN {X 0,Y 253.778,Z 642.825,A -85,B 0,C 180,E1 177.119,E2 177.119} C_VEL
LIN {X 0,Y 240.512,Z 660.253,A -85,B 0,C 180,E1 176.113,E2 176.113} C_VEL
LIN {X 0,Y 225.875,Z 677.131,A -85,B 0,C 180,E1 174.846,E2 174.846} C_VEL
LIN {X 0,Y 210.401,Z 692.551,A -85,B 0,C 180,E1 173.302,E2 173.302} C_VEL
LIN {X 0,Y 193.21,Z 707.552,A -85,B 0,C 180,E1 171.262,E2 171.262} C_VEL
LIN {X 0,Y 175.384,Z 721.155,A -85,B 0,C 180,E1 168.677,E2 168.677} C_VEL
LIN {X 0,Y 157.086,Z 733.143,A -85,B 0,C 180,E1 165.342,E2 165.342} C_VEL
LIN {X 0,Y 138.591,Z 743.717,A -85,B 0,C 180,E1 160.921,E2 160.921} C_VEL
LIN {X 0,Y 121.128,Z 752.442,A -85,B 0,C 180,E1 155.227,E2 155.227} C_VEL
LIN {X 0,Y 104.448,Z 759.591,A -85,B 0,C 180,E1 147.392,E2 147.392} C_VEL
LIN {X 0,Y 89.084,Z 765.46,A -85,B 0,C 180,E1 135.902,E2 135.902} C_VEL
LIN {X 0,Y 78.816,Z 769.174,A -85,B 0,C 180,E1 122.194,E2 122.194} C_VEL
LIN {X 0,Y 73.424,Z 771.119,A -85,B 0,C 180,E1 106.616,E2 106.616} C_VEL
LIN {X 0,Y 72.173,Z 771.743,A -85,B 0,C 180,E1 93.972,E2 93.972} C_VEL
LIN {X 0,Y 72.256,Z 771.69,A -85,B 0,C 180,E1 83.644,E2 83.644} C_VEL
LIN {X 0,Y 74.074,Z 770.893,A -85,B 0,C 180,E1 70.279,E2 70.279} C_VEL
LIN {X 0,Y 80.726,Z 768.47,A -85,B 0,C 180,E1 54.401,E2 54.401} C_VEL
LIN {X 0,Y 91.933,Z 764.536,A -85,B 0,C 180,E1 41.373,E2 41.373} C_VEL
LIN {X 0,Y 106.54,Z 758.806,A -85,B 0,C 180,E1 31.351,E2 31.351} C_VEL
LIN {X 0,Y 124.294,Z 750.987,A -85,B 0,C 180,E1 23.505,E2 23.505} C_VEL
LIN {X 0,Y 141.992,Z 742.055,A -85,B 0,C 180,E1 18.086,E2 18.086} C_VEL
LIN {X 0,Y 159.744,Z 731.615,A -85,B 0,C 180,E1 14.038,E2 14.038} C_VEL
LIN {X 0,Y 178.129,Z 719.295,A -85,B 0,C 180,E1 10.806,E2 10.806} C_VEL
LIN {X 0,Y 194.12,Z 707.008,A -85,B 0,C 180,E1 8.541,E2 8.541} C_VEL
LIN {X 0,Y 211.33,Z 691.893,A -85,B 0,C 180,E1 6.518,E2 6.518} C_VEL
LIN {X 0,Y 227.307,Z 675.873,A -85,B 0,C 180,E1 4.943,E2 4.943} C_VEL
LIN {X 0,Y 241.961,Z 658.784,A -85,B 0,C 180,E1 3.693,E2 3.693} C_VEL
LIN {X 0,Y 256.226,Z 639.596,A -85,B 0,C 180,E1 2.629,E2 2.629} C_VEL
LIN {X 0,Y 265.477,Z 625.321,A -85,B 0,C 180,E1 2.001,E2 2.001} C_VEL
LIN {X 0,Y 252.908,Z 644.464,A -85,B 0,C 180,E1 1.133,E2 1.133} C_VEL
LIN {X 0,Y 238.959,Z 662.563,A -85,B 0,C 180,E1 0.059,E2 0.059} C_VEL
LIN {X 0,Y 223.152,Z 680.407,A -85,B 0,C 180,E1 -1.34,E2 -1.34} C_VEL
LIN {X 0,Y 217.709,Z 686.005,A -85,B 0,C 180,E1 -1.601,E2 -1.601} C_VEL
LIN {X 0,Y 202.844,Z 699.484,A -85,B 0,C 180,E1 -1.403,E2 -1.403} C_VEL
LIN {X 0,Y 197.058,Z 704.429,A -85,B 0,C 180,E1 -1.725,E2 -1.725} C_VEL
LIN {X 0,Y 179.379,Z 718.261,A -85,B 0,C 180,E1 -3.873,E2 -3.873} C_VEL
LIN {X 0,Y 161.057,Z 730.894,A -85,B 0,C 180,E1 -6.651,E2 -6.651} C_VEL
LIN {X 0,Y 142.279,Z 742.107,A -85,B 0,C 180,E1 -10.323,E2 -10.323} C_VEL
LIN {X 0,Y 123.362,Z 751.963,A -85,B 0,C 180,E1 -15.318,E2 -15.318} C_VEL
LIN {X 0,Y 104.858,Z 760.433,A -85,B 0,C 180,E1 -22.346,E2 -22.346} C_VEL
LIN {X 0,Y 88.425,Z 766.949,A -85,B 0,C 180,E1 -32.001,E2 -32.001} C_VEL
LIN {X 0,Y 74.725,Z 771.993,A -85,B 0,C 180,E1 -45.912,E2 -45.912} C_VEL
LIN {X 0,Y 66.987,Z 774.947,A -85,B 0,C 180,E1 -61.718,E2 -61.718} C_VEL
LIN {X 0,Y 64.135,Z 776.496,A -85,B 0,C 180,E1 -79.218,E2 -79.218} C_VEL
LIN {X 0,Y 64.124,Z 776.803,A -85,B 0,C 180,E1 -90,E2 -90} C_VEL
LIN {X 0,Y 64.175,Z 776.463,A -85,B 0,C 180,E1 -101.685,E2 -101.685} C_VEL
LIN {X 0,Y 67.326,Z 774.767,A -85,B 0,C 180,E1 -119.345,E2 -119.345} C_VEL
LIN {X 0,Y 75.225,Z 771.786,A -85,B 0,C 180,E1 -134.784,E2 -134.784} C_VEL
LIN {X 0,Y 89.108,Z 766.623,A -85,B 0,C 180,E1 -148.512,E2 -148.512} C_VEL
LIN {X 0,Y 105.658,Z 760.011,A -85,B 0,C 180,E1 -158.028,E2 -158.028} C_VEL
LIN {X 0,Y 123.359,Z 751.87,A -85,B 0,C 180,E1 -164.688,E2 -164.688} C_VEL
LIN {X 0,Y 143.572,Z 741.25,A -85,B 0,C 180,E1 -169.974,E2 -169.974} C_VEL
LIN {X 0,Y 162.008,Z 730.169,A -85,B 0,C 180,E1 -173.518,E2 -173.518} C_VEL
LIN {X 0,Y 180.352,Z 717.377,A -85,B 0,C 180,E1 -176.265,E2 -176.265} C_VEL
LIN {X 0,Y 199.034,Z 702.504,A -85,B 0,C 180,E1 -178.5,E2 -178.5} C_VEL
LIN {X 0,Y 215.964,Z 687.087,A -85,B 0,C 180,E1 -180.167,E2 -180.167} C_VEL
LIN {X 0,Y 231.657,Z 670.531,A -85,B 0,C 180,E1 -181.484,E2 -181.484} C_VEL
LIN {X 0,Y 238.953,Z 662.043,A -85,B 0,C 180,E1 -182.052,E2 -182.052} C_VEL
LIN {X 0,Y 222.833,Z 679.993,A -85,B 0,C 180,E1 -183.308,E2 -183.308} C_VEL
LIN {X 0,Y 206.686,Z 695.636,A -85,B 0,C 180,E1 -184.786,E2 -184.786} C_VEL
LIN {X 0,Y 189.253,Z 710.156,A -85,B 0,C 180,E1 -186.68,E2 -186.68} C_VEL
LIN {X 0,Y 170.18,Z 723.974,A -85,B 0,C 180,E1 -189.242,E2 -189.242} C_VEL
LIN {X 0,Y 151.533,Z 735.693,A -85,B 0,C 180,E1 -192.441,E2 -192.441} C_VEL
LIN {X 0,Y 132.588,Z 745.812,A -85,B 0,C 180,E1 -196.725,E2 -196.725} C_VEL
LIN {X 0,Y 113.218,Z 754.708,A -85,B 0,C 180,E1 -202.867,E2 -202.867} C_VEL
LIN {X 0,Y 96.538,Z 761.351,A -85,B 0,C 180,E1 -210.726,E2 -210.726} C_VEL
LIN {X 0,Y 81.787,Z 766.348,A -85,B 0,C 180,E1 -221.779,E2 -221.779} C_VEL
LIN {X 0,Y 70.088,Z 770.013,A -85,B 0,C 180,E1 -238.142,E2 -238.142} C_VEL
LIN {X 0,Y 65.24,Z 771.6,A -85,B 0,C 180,E1 -253.987,E2 -253.987} C_VEL
LIN {X 0,Y 64.143,Z 772.097,A -85,B 0,C 180,E1 -268.214,E2 -268.214} C_VEL
LIN {X 0,Y 64.552,Z 771.904,A -85,B 0,C 180,E1 -280.712,E2 -280.712} C_VEL
LIN {X 0,Y 68.691,Z 770.475,A -85,B 0,C 180,E1 -298.707,E2 -298.707} C_VEL
LIN {X 0,Y 77.775,Z 767.706,A -85,B 0,C 180,E1 -313.963,E2 -313.963} C_VEL
LIN {X 0,Y 91.465,Z 763.147,A -85,B 0,C 180,E1 -326.179,E2 -326.179} C_VEL
LIN {X 0,Y 108.023,Z 756.985,A -85,B 0,C 180,E1 -335.102,E2 -335.102} C_VEL
LIN {X 0,Y 125.833,Z 749.184,A -85,B 0,C 180,E1 -341.467,E2 -341.467} C_VEL
LIN {X 0,Y 145.088,Z 739.369,A -85,B 0,C 180,E1 -346.327,E2 -346.327} C_VEL
LIN {X 0,Y 163.563,Z 728.518,A -85,B 0,C 180,E1 -349.79,E2 -349.79} C_VEL
LIN {X 0,Y 181.549,Z 716.163,A -85,B 0,C 180,E1 -352.437,E2 -352.437} C_VEL
LIN {X 0,Y 199.854,Z 701.731,A -85,B 0,C 180,E1 -354.598,E2 -354.598} C_VEL
LIN {X 0,Y 216.436,Z 686.747,A -85,B 0,C 180,E1 -356.213,E2 -356.213} C_VEL
LIN {X 0,Y 232.177,Z 670.206,A -85,B 0,C 180,E1 -357.524,E2 -357.524} C_VEL
LIN {X 0,Y 238.548,Z 662.852,A -85,B 0,C 180,E1 -358.005,E2 -358.005} C_VEL
LIN {X 0,Y 222.929,Z 680.234,A -85,B 0,C 180,E1 -359.229,E2 -359.229} C_VEL
LIN {X 0,Y 206.98,Z 695.785,A -85,B 0,C 180,E1 -360.688,E2 -360.688} C_VEL
LIN {X 0,Y 197.058,Z 704.429,A -85,B 0,C 180,E1 -361.725,E2 -361.725} C_VEL
LIN {X 0,Y 191.13,Z 709.306,A -85,B 0,C 180,E1 -362.082,E2 -362.082} C_VEL
LIN {X 0,Y 174.78,Z 721.061,A -85,B 0,C 180,E1 -362.056,E2 -362.056} C_VEL
LIN {X 0,Y 168.435,Z 725.273,A -85,B 0,C 180,E1 -362.531,E2 -362.531} C_VEL
LIN {X 0,Y 149.636,Z 737.032,A -85,B 0,C 180,E1 -365.387,E2 -365.387} C_VEL
LIN {X 0,Y 129.716,Z 747.66,A -85,B 0,C 180,E1 -369.388,E2 -369.388} C_VEL
LIN {X 0,Y 109.75,Z 756.852,A -85,B 0,C 180,E1 -375.058,E2 -375.058} C_VEL
LIN {X 0,Y 91.241,Z 764.233,A -85,B 0,C 180,E1 -383.003,E2 -383.003} C_VEL
LIN {X 0,Y 75.13,Z 769.717,A -85,B 0,C 180,E1 -394.402,E2 -394.402} C_VEL
LIN {X 0,Y 62.464,Z 773.782,A -85,B 0,C 180,E1 -411.657,E2 -411.657} C_VEL
LIN {X 0,Y 57.041,Z 775.704,A -85,B 0,C 180,E1 -429.478,E2 -429.478} C_VEL
LIN {X 0,Y 56.066,Z 776.397,A -85,B 0,C 180,E1 -444.884,E2 -444.884} C_VEL
LIN {X 0,Y 56.082,Z 776.438,A -85,B 0,C 180,E1 -453.282,E2 -453.282} C_VEL
LIN {X 0,Y 56.753,Z 775.84,A -85,B 0,C 180,E1 -468.488,E2 -468.488} C_VEL
LIN {X 0,Y 61.362,Z 774.096,A -85,B 0,C 180,E1 -485.915,E2 -485.915} C_VEL
LIN {X 0,Y 72.569,Z 770.543,A -85,B 0,C 180,E1 -503.045,E2 -503.045} C_VEL
LIN {X 0,Y 87.322,Z 765.519,A -85,B 0,C 180,E1 -514.763,E2 -514.763} C_VEL
LIN {X 0,Y 106.252,Z 758.236,A -85,B 0,C 180,E1 -523.703,E2 -523.703} C_VEL
LIN {X 0,Y 125.083,Z 749.889,A -85,B 0,C 180,E1 -529.477,E2 -529.477} C_VEL
LIN {X 0,Y 144.831,Z 739.564,A -85,B 0,C 180,E1 -533.77,E2 -533.77} C_VEL
LIN {X 0,Y 165.193,Z 727.261,A -85,B 0,C 180,E1 -537.034,E2 -537.034} C_VEL
LIN {X 0,Y 184.086,Z 714.109,A -85,B 0,C 180,E1 -539.378,E2 -539.378} C_VEL
LIN {X 0,Y 202.008,Z 699.581,A -85,B 0,C 180,E1 -541.177,E2 -541.177} C_VEL
LIN {X 0,Y 211.851,Z 690.727,A -85,B 0,C 180,E1 -542.054,E2 -542.054} C_VEL
LIN {X 0,Y 195.338,Z 705.157,A -85,B 0,C 180,E1 -543.533,E2 -543.533} C_VEL
LIN {X 0,Y 177.765,Z 718.358,A -85,B 0,C 180,E1 -545.42,E2 -545.42} C_VEL
LIN {X 0,Y 158.52,Z 730.948,A -85,B 0,C 180,E1 -548.011,E2 -548.011} C_VEL
LIN {X 0,Y 139.682,Z 741.553,A -85,B 0,C 180,E1 -551.294,E2 -551.294} C_VEL
LIN {X 0,Y 120.533,Z 750.685,A -85,B 0,C 180,E1 -555.798,E2 -555.798} C_VEL
LIN {X 0,Y 101.527,Z 758.432,A -85,B 0,C 180,E1 -562.226,E2 -562.226} C_VEL
LIN {X 0,Y 84.981,Z 764.105,A -85,B 0,C 180,E1 -570.811,E2 -570.811} C_VEL
LIN {X 0,Y 69.82,Z 768.558,A -85,B 0,C 180,E1 -584.275,E2 -584.275} C_VEL
LIN {X 0,Y 59.988,Z 771.264,A -85,B 0,C 180,E1 -602.181,E2 -602.181} C_VEL
LIN {X 0,Y 56.416,Z 772.246,A -85,B 0,C 180,E1 -620.822,E2 -620.822} C_VEL
LIN {X 0,Y 56.161,Z 772.374,A -85,B 0,C 180,E1 -633.062,E2 -633.062} C_VEL
LIN {X 0,Y 57.696,Z 771.852,A -85,B 0,C 180,E1 -649.224,E2 -649.224} C_VEL
LIN {X 0,Y 64.175,Z 770.132,A -85,B 0,C 180,E1 -667.417,E2 -667.417} C_VEL
LIN {X 0,Y 77.241,Z 766.495,A -85,B 0,C 180,E1 -683.454,E2 -683.454} C_VEL
LIN {X 0,Y 93.36,Z 761.453,A -85,B 0,C 180,E1 -694.105,E2 -694.105} C_VEL
LIN {X 0,Y 111.685,Z 754.538,A -85,B 0,C 180,E1 -701.61,E2 -701.61} C_VEL
LIN {X 0,Y 131.342,Z 745.791,A -85,B 0,C 180,E1 -707.005,E2 -707.005} C_VEL
LIN {X 0,Y 149.952,Z 736.144,A -85,B 0,C 180,E1 -710.686,E2 -710.686} C_VEL
LIN {X 0,Y 169.037,Z 724.458,A -85,B 0,C 180,E1 -713.564,E2 -713.564} C_VEL
LIN {X 0,Y 188.461,Z 710.691,A -85,B 0,C 180,E1 -715.853,E2 -715.853} C_VEL
LIN {X 0,Y 206.155,Z 696.216,A -85,B 0,C 180,E1 -717.537,E2 -717.537} C_VEL
LIN {X 0,Y 211.56,Z 691.234,A -85,B 0,C 180,E1 -718.009,E2 -718.009} C_VEL
LIN {X 0,Y 193.972,Z 706.553,A -85,B 0,C 180,E1 -719.594,E2 -719.594} C_VEL
LIN {X 0,Y 176.035,Z 720.079,A -85,B 0,C 180,E1 -721.56,E2 -721.56} C_VEL
LIN {X 0,Y 168.435,Z 725.273,A -85,B 0,C 180,E1 -722.531,E2 -722.531} C_VEL
LIN {X 0,Y 161.992,Z 729.457,A -85,B 0,C 180,E1 -723.056,E2 -723.056} C_VEL
LIN {X 0,Y 144.461,Z 739.289,A -85,B 0,C 180,E1 -723.293,E2 -723.293} C_VEL
LIN {X 0,Y 137.794,Z 742.811,A -85,B 0,C 180,E1 -723.978,E2 -723.978} C_VEL
LIN {X 0,Y 118.132,Z 752.188,A -85,B 0,C 180,E1 -728.009,E2 -728.009} C_VEL
LIN {X 0,Y 97.902,Z 760.459,A -85,B 0,C 180,E1 -734.023,E2 -734.023} C_VEL
LIN {X 0,Y 79.999,Z 766.606,A -85,B 0,C 180,E1 -742.354,E2 -742.354} C_VEL
LIN {X 0,Y 63.197,Z 771.562,A -85,B 0,C 180,E1 -756.21,E2 -756.21} C_VEL
LIN {X 0,Y 52.329,Z 774.583,A -85,B 0,C 180,E1 -775.243,E2 -775.243} C_VEL
LIN {X 0,Y 48.178,Z 775.966,A -85,B 0,C 180,E1 -798.023,E2 -798.023} C_VEL
LIN {X 0,Y 48.112,Z 776.201,A -85,B 0,C 180,E1 -811.191,E2 -811.191} C_VEL
LIN {X 0,Y 48.507,Z 775.838,A -85,B 0,C 180,E1 -826.772,E2 -826.772} C_VEL
LIN {X 0,Y 53.994,Z 774.043,A -85,B 0,C 180,E1 -849.02,E2 -849.02} C_VEL
LIN {X 0,Y 66.5,Z 770.666,A -85,B 0,C 180,E1 -867.348,E2 -867.348} C_VEL
LIN {X 0,Y 83.262,Z 765.482,A -85,B 0,C 180,E1 -879.495,E2 -879.495} C_VEL
LIN {X 0,Y 103.298,Z 758.296,A -85,B 0,C 180,E1 -887.848,E2 -887.848} C_VEL
LIN {X 0,Y 123.824,Z 749.581,A -85,B 0,C 180,E1 -893.304,E2 -893.304} C_VEL
LIN {X 0,Y 144.162,Z 739.252,A -85,B 0,C 180,E1 -897.086,E2 -897.086} C_VEL
LIN {X 0,Y 165.484,Z 726.606,A -85,B 0,C 180,E1 -900.001,E2 -900.001} C_VEL
LIN {X 0,Y 184.077,Z 713.857,A -85,B 0,C 180,E1 -901.967,E2 -901.967} C_VEL
LIN {X 0,Y 184.714,Z 713.372,A -85,B 0,C 180,E1 -902.063,E2 -902.063} C_VEL
LIN {X 0,Y 166.373,Z 725.849,A -85,B 0,C 180,E1 -903.98,E2 -903.98} C_VEL
LIN {X 0,Y 146.94,Z 737.318,A -85,B 0,C 180,E1 -906.571,E2 -906.571} C_VEL
LIN {X 0,Y 127.892,Z 746.869,A -85,B 0,C 180,E1 -909.924,E2 -909.924} C_VEL
LIN {X 0,Y 107.604,Z 755.424,A -85,B 0,C 180,E1 -914.908,E2 -914.908} C_VEL
LIN {X 0,Y 88.443,Z 762.198,A -85,B 0,C 180,E1 -922.03,E2 -922.03} C_VEL
LIN {X 0,Y 71.208,Z 767.142,A -85,B 0,C 180,E1 -932.599,E2 -932.599} C_VEL
LIN {X 0,Y 56.921,Z 770.606,A -85,B 0,C 180,E1 -949.465,E2 -949.465} C_VEL
LIN {X 0,Y 49.706,Z 772.25,A -85,B 0,C 180,E1 -970.004,E2 -970.004} C_VEL
LIN {X 0,Y 48.151,Z 772.701,A -85,B 0,C 180,E1 -988.81,E2 -988.81} C_VEL
LIN {X 0,Y 48.98,Z 772.47,A -85,B 0,C 180,E1 -1005.389,E2 -1005.389} C_VEL
LIN {X 0,Y 55.449,Z 770.957,A -85,B 0,C 180,E1 -1027.812,E2 -1027.812} C_VEL
LIN {X 0,Y 68.347,Z 767.987,A -85,B 0,C 180,E1 -1045.006,E2 -1045.006} C_VEL
LIN {X 0,Y 85.239,Z 763.206,A -85,B 0,C 180,E1 -1056.494,E2 -1056.494} C_VEL
LIN {X 0,Y 105.771,Z 756.209,A -85,B 0,C 180,E1 -1064.619,E2 -1064.619} C_VEL
LIN {X 0,Y 125.049,Z 748.327,A -85,B 0,C 180,E1 -1069.561,E2 -1069.561} C_VEL
LIN {X 0,Y 144.992,Z 738.464,A -85,B 0,C 180,E1 -1073.211,E2 -1073.211} C_VEL
LIN {X 0,Y 165.378,Z 726.643,A -85,B 0,C 180,E1 -1075.983,E2 -1075.983} C_VEL
LIN {X 0,Y 184.48,Z 713.746,A -85,B 0,C 180,E1 -1078.005,E2 -1078.005} C_VEL
LIN {X 0,Y 165.562,Z 726.711,A -85,B 0,C 180,E1 -1079.999,E2 -1079.999} C_VEL
LIN {X 0,Y 144.163,Z 739.373,A -85,B 0,C 180,E1 -1082.922,E2 -1082.922} C_VEL
LIN {X 0,Y 137.794,Z 742.811,A -85,B 0,C 180,E1 -1083.978,E2 -1083.978} C_VEL
LIN {X 0,Y 131.048,Z 746.208,A -85,B 0,C 180,E1 -1084.749,E2 -1084.749} C_VEL
LIN {X 0,Y 111.508,Z 754.417,A -85,B 0,C 180,E1 -1085.58,E2 -1085.58} C_VEL
LIN {X 0,Y 105.541,Z 756.66,A -85,B 0,C 180,E1 -1086.574,E2 -1086.574} C_VEL
LIN {X 0,Y 85.178,Z 763.904,A -85,B 0,C 180,E1 -1093.027,E2 -1093.027} C_VEL
LIN {X 0,Y 66.317,Z 769.328,A -85,B 0,C 180,E1 -1103.123,E2 -1103.123} C_VEL
LIN {X 0,Y 50.085,Z 773.275,A -85,B 0,C 180,E1 -1120.661,E2 -1120.661} C_VEL
LIN {X 0,Y 41.844,Z 775.186,A -85,B 0,C 180,E1 -1143,E2 -1143} C_VEL
LIN {X 0,Y 40.076,Z 775.839,A -85,B 0,C 180,E1 -1164.273,E2 -1164.273} C_VEL
LIN {X 0,Y 40.078,Z 775.86,A -85,B 0,C 180,E1 -1174.292,E2 -1174.292} C_VEL
LIN {X 0,Y 41.592,Z 775.246,A -85,B 0,C 180,E1 -1195.639,E2 -1195.639} C_VEL
LIN {X 0,Y 49.508,Z 773.372,A -85,B 0,C 180,E1 -1218.35,E2 -1218.35} C_VEL
LIN {X 0,Y 65.519,Z 769.499,A -85,B 0,C 180,E1 -1236.292,E2 -1236.292} C_VEL
LIN {X 0,Y 83.378,Z 764.377,A -85,B 0,C 180,E1 -1246.242,E2 -1246.242} C_VEL
LIN {X 0,Y 103.761,Z 757.257,A -85,B 0,C 180,E1 -1252.975,E2 -1252.975} C_VEL
LIN {X 0,Y 124.11,Z 748.816,A -85,B 0,C 180,E1 -1257.37,E2 -1257.37} C_VEL
LIN {X 0,Y 143.979,Z 738.939,A -85,B 0,C 180,E1 -1260.42,E2 -1260.42} C_VEL
LIN {X 0,Y 157.497,Z 731.329,A -85,B 0,C 180,E1 -1262.045,E2 -1262.045} C_VEL
LIN {X 0,Y 138.393,Z 741.662,A -85,B 0,C 180,E1 -1264.447,E2 -1264.447} C_VEL
LIN {X 0,Y 118.092,Z 750.89,A -85,B 0,C 180,E1 -1267.87,E2 -1267.87} C_VEL
LIN {X 0,Y 98.364,Z 758.439,A -85,B 0,C 180,E1 -1272.632,E2 -1272.632} C_VEL
LIN {X 0,Y 78.415,Z 764.549,A -85,B 0,C 180,E1 -1280.139,E2 -1280.139} C_VEL
LIN {X 0,Y 59.579,Z 769.152,A -85,B 0,C 180,E1 -1292.957,E2 -1292.957} C_VEL
LIN {X 0,Y 46.263,Z 771.854,A -85,B 0,C 180,E1 -1312.761,E2 -1312.761} C_VEL
LIN {X 0,Y 40.644,Z 772.83,A -85,B 0,C 180,E1 -1337.209,E2 -1337.209} C_VEL
LIN {X 0,Y 40.188,Z 772.955,A -85,B 0,C 180,E1 -1354.28,E2 -1354.28} C_VEL
LIN {X 0,Y 42.763,Z 772.439,A -85,B 0,C 180,E1 -1376.374,E2 -1376.374} C_VEL
LIN {X 0,Y 52.184,Z 770.721,A -85,B 0,C 180,E1 -1398.351,E2 -1398.351} C_VEL
LIN {X 0,Y 68.712,Z 767.101,A -85,B 0,C 180,E1 -1414.443,E2 -1414.443} C_VEL
LIN {X 0,Y 87.451,Z 762.05,A -85,B 0,C 180,E1 -1423.816,E2 -1423.816} C_VEL
LIN {X 0,Y 107.642,Z 755.133,A -85,B 0,C 180,E1 -1429.925,E2 -1429.925} C_VEL
LIN {X 0,Y 129.207,Z 746.139,A -85,B 0,C 180,E1 -1434.226,E2 -1434.226} C_VEL
LIN {X 0,Y 149.171,Z 736.22,A -85,B 0,C 180,E1 -1437.059,E2 -1437.059} C_VEL
LIN {X 0,Y 157.068,Z 731.719,A -85,B 0,C 180,E1 -1438.01,E2 -1438.01} C_VEL
LIN {X 0,Y 136.983,Z 742.754,A -85,B 0,C 180,E1 -1440.556,E2 -1440.556} C_VEL
LIN {X 0,Y 116.284,Z 752.301,A -85,B 0,C 180,E1 -1444.139,E2 -1444.139} C_VEL
LIN {X 0,Y 105.541,Z 756.66,A -85,B 0,C 180,E1 -1446.574,E2 -1446.574} C_VEL
LIN {X 0,Y 98.537,Z 759.265,A -85,B 0,C 180,E1 -1447.826,E2 -1447.826} C_VEL
LIN {X 0,Y 78.907,Z 765.039,A -85,B 0,C 180,E1 -1449.771,E2 -1449.771} C_VEL
LIN {X 0,Y 72.384,Z 766.823,A -85,B 0,C 180,E1 -1451.673,E2 -1451.673} C_VEL
LIN {X 0,Y 53.405,Z 771.3,A -85,B 0,C 180,E1 -1463.458,E2 -1463.458} C_VEL
LIN {X 0,Y 38.334,Z 774.273,A -85,B 0,C 180,E1 -1485.233,E2 -1485.233} C_VEL
LIN {X 0,Y 32.361,Z 775.405,A -85,B 0,C 180,E1 -1513.855,E2 -1513.855} C_VEL
LIN {X 0,Y 32.132,Z 775.639,A -85,B 0,C 180,E1 -1530,E2 -1530} C_VEL
LIN {X 0,Y 32.818,Z 775.312,A -85,B 0,C 180,E1 -1551.444,E2 -1551.444} C_VEL
LIN {X 0,Y 41.815,Z 773.567,A -85,B 0,C 180,E1 -1582.098,E2 -1582.098} C_VEL
LIN {X 0,Y 57.504,Z 770.407,A -85,B 0,C 180,E1 -1599.869,E2 -1599.869} C_VEL
LIN {X 0,Y 77.196,Z 765.379,A -85,B 0,C 180,E1 -1610.308,E2 -1610.308} C_VEL
LIN {X 0,Y 98.163,Z 758.775,A -85,B 0,C 180,E1 -1616.535,E2 -1616.535} C_VEL
LIN {X 0,Y 118.984,Z 750.639,A -85,B 0,C 180,E1 -1620.497,E2 -1620.497} C_VEL
LIN {X 0,Y 129.689,Z 745.849,A -85,B 0,C 180,E1 -1622.085,E2 -1622.085} C_VEL
LIN {X 0,Y 108.47,Z 754.647,A -85,B 0,C 180,E1 -1625.438,E2 -1625.438} C_VEL
LIN {X 0,Y 88.363,Z 761.383,A -85,B 0,C 180,E1 -1630.133,E2 -1630.133} C_VEL
LIN {X 0,Y 67.371,Z 766.946,A -85,B 0,C 180,E1 -1638.232,E2 -1638.232} C_VEL
LIN {X 0,Y 49.236,Z 770.68,A -85,B 0,C 180,E1 -1651.872,E2 -1651.872} C_VEL
LIN {X 0,Y 36.124,Z 772.652,A -85,B 0,C 180,E1 -1676.389,E2 -1676.389} C_VEL
LIN {X 0,Y 32.268,Z 773.22,A -85,B 0,C 180,E1 -1702.88,E2 -1702.88} C_VEL
LIN {X 0,Y 32.432,Z 773.186,A -85,B 0,C 180,E1 -1720.66,E2 -1720.66} C_VEL
LIN {X 0,Y 36.985,Z 772.547,A -85,B 0,C 180,E1 -1746.494,E2 -1746.494} C_VEL
LIN {X 0,Y 50.84,Z 770.403,A -85,B 0,C 180,E1 -1769.918,E2 -1769.918} C_VEL
LIN {X 0,Y 69.106,Z 766.606,A -85,B 0,C 180,E1 -1782.724,E2 -1782.724} C_VEL
LIN {X 0,Y 90.228,Z 760.879,A -85,B 0,C 180,E1 -1790.477,E2 -1790.477} C_VEL
LIN {X 0,Y 111.375,Z 753.675,A -85,B 0,C 180,E1 -1795.178,E2 -1795.178} C_VEL
LIN {X 0,Y 129.546,Z 746.031,A -85,B 0,C 180,E1 -1797.995,E2 -1797.995} C_VEL
LIN {X 0,Y 108.014,Z 755.208,A -85,B 0,C 180,E1 -1801.402,E2 -1801.402} C_VEL
LIN {X 0,Y 87.505,Z 762.376,A -85,B 0,C 180,E1 -1806.247,E2 -1806.247} C_VEL
LIN {X 0,Y 72.384,Z 766.823,A -85,B 0,C 180,E1 -1811.673,E2 -1811.673} C_VEL
LIN {X 0,Y 65.395,Z 768.556,A -85,B 0,C 180,E1 -1814.087,E2 -1814.087} C_VEL
LIN {X 0,Y 44.722,Z 772.213,A -85,B 0,C 180,E1 -1820.472,E2 -1820.472} C_VEL
LIN {X 0,Y 39.566,Z 772.934,A -85,B 0,C 180,E1 -1824.858,E2 -1824.858} C_VEL
LIN {X 0,Y 26.851,Z 774.82,A -85,B 0,C 180,E1 -1853.432,E2 -1853.432} C_VEL
LIN {X 0,Y 24.1,Z 775.333,A -85,B 0,C 180,E1 -1887.622,E2 -1887.622} C_VEL
LIN {X 0,Y 24.488,Z 775.134,A -85,B 0,C 180,E1 -1909.064,E2 -1909.064} C_VEL
LIN {X 0,Y 32.992,Z 773.957,A -85,B 0,C 180,E1 -1944.908,E2 -1944.908} C_VEL
LIN {X 0,Y 50.667,Z 770.96,A -85,B 0,C 180,E1 -1965.224,E2 -1965.224} C_VEL
LIN {X 0,Y 71.97,Z 766.236,A -85,B 0,C 180,E1 -1975.22,E2 -1975.22} C_VEL
LIN {X 0,Y 93.496,Z 759.943,A -85,B 0,C 180,E1 -1980.614,E2 -1980.614} C_VEL
LIN {X 0,Y 101.552,Z 757.183,A -85,B 0,C 180,E1 -1982.102,E2 -1982.102} C_VEL
LIN {X 0,Y 78.57,Z 764.073,A -85,B 0,C 180,E1 -1986.984,E2 -1986.984} C_VEL
LIN {X 0,Y 57.898,Z 768.824,A -85,B 0,C 180,E1 -1994.748,E2 -1994.748} C_VEL
LIN {X 0,Y 39.156,Z 771.812,A -85,B 0,C 180,E1 -2009.754,E2 -2009.754} C_VEL
LIN {X 0,Y 26.47,Z 773.341,A -85,B 0,C 180,E1 -2040.591,E2 -2040.591} C_VEL
LIN {X 0,Y 24.169,Z 773.592,A -85,B 0,C 180,E1 -2070,E2 -2070} C_VEL
LIN {X 0,Y 27.252,Z 773.277,A -85,B 0,C 180,E1 -2103.389,E2 -2103.389} C_VEL
LIN {X 0,Y 40.696,Z 771.63,A -85,B 0,C 180,E1 -2132.185,E2 -2132.185} C_VEL
LIN {X 0,Y 60.621,Z 768.29,A -85,B 0,C 180,E1 -2146.679,E2 -2146.679} C_VEL
LIN {X 0,Y 81.453,Z 763.407,A -85,B 0,C 180,E1 -2153.862,E2 -2153.862} C_VEL
LIN {X 0,Y 101.435,Z 757.319,A -85,B 0,C 180,E1 -2157.98,E2 -2157.98} C_VEL
LIN {X 0,Y 78.09,Z 764.632,A -85,B 0,C 180,E1 -2162.947,E2 -2162.947} C_VEL
LIN {X 0,Y 56.565,Z 769.888,A -85,B 0,C 180,E1 -2171.21,E2 -2171.21} C_VEL
LIN {X 0,Y 39.566,Z 772.934,A -85,B 0,C 180,E1 -2184.858,E2 -2184.858} C_VEL
LIN {X 0,Y 32.89,Z 773.88,A -85,B 0,C 180,E1 -2192.605,E2 -2192.605} C_VEL
LIN {X 0,Y 21.673,Z 774.776,A -85,B 0,C 180,E1 -2210.587,E2 -2210.587} C_VEL
LIN {X 0,Y 16.108,Z 775.035,A -85,B 0,C 180,E1 -2245.091,E2 -2245.091} C_VEL
LIN {X 0,Y 16.11,Z 775.053,A -85,B 0,C 180,E1 -2249.101,E2 -2249.101} C_VEL
LIN {X 0,Y 18.619,Z 774.719,A -85,B 0,C 180,E1 -2290.119,E2 -2290.119} C_VEL
LIN {X 0,Y 34.674,Z 772.904,A -85,B 0,C 180,E1 -2324.961,E2 -2324.961} C_VEL
LIN {X 0,Y 55.061,Z 769.631,A -85,B 0,C 180,E1 -2337.096,E2 -2337.096} C_VEL
LIN {X 0,Y 72.568,Z 765.717,A -85,B 0,C 180,E1 -2342.087,E2 -2342.087} C_VEL
LIN {X 0,Y 50.174,Z 770.112,A -85,B 0,C 180,E1 -2349.175,E2 -2349.175} C_VEL
LIN {X 0,Y 29.811,Z 772.809,A -85,B 0,C 180,E1 -2365.102,E2 -2365.102} C_VEL
LIN {X 0,Y 17.553,Z 773.725,A -85,B 0,C 180,E1 -2402.891,E2 -2402.891} C_VEL
LIN {X 0,Y 16.234,Z 773.849,A -85,B 0,C 180,E1 -2437.076,E2 -2437.076} C_VEL
LIN {X 0,Y 22.922,Z 773.384,A -85,B 0,C 180,E1 -2481.734,E2 -2481.734} C_VEL
LIN {X 0,Y 39.398,Z 771.714,A -85,B 0,C 180,E1 -2504.654,E2 -2504.654} C_VEL
LIN {X 0,Y 61.221,Z 768.191,A -85,B 0,C 180,E1 -2515.02,E2 -2515.02} C_VEL
LIN {X 0,Y 72.416,Z 765.82,A -85,B 0,C 180,E1 -2517.953,E2 -2517.953} C_VEL
LIN {X 0,Y 50.175,Z 770.527,A -85,B 0,C 180,E1 -2524.907,E2 -2524.907} C_VEL
LIN {X 0,Y 29.885,Z 773.595,A -85,B 0,C 180,E1 -2540.486,E2 -2540.486} C_VEL
LIN {X 0,Y 17.064,Z 774.84,A -85,B 0,C 180,E1 -2581.501,E2 -2581.501} C_VEL
LIN {X 0,Y 16.11,Z 775.053,A -85,B 0,C 180,E1 -2609.101,E2 -2609.101} C_VEL
LIN {X 0,Y 16.349,Z 775.045,A -85,B 0,C 180,E1 -2628.419,E2 -2628.419} C_VEL
LIN {X 0,Y 17.349,Z 774.804,A -85,B 0,C 180,E1 -2652.848,E2 -2652.848} C_VEL
LIN {X 0,Y 27.435,Z 773.371,A -85,B 0,C 180,E1 -2693.812,E2 -2693.812} C_VEL
LIN {X 0,Y 32.076,Z 772.779,A -85,B 0,C 180,E1 -2698.042,E2 -2698.042} C_VEL
LIN {X 0,Y 41.507,Z 771.61,A -85,B 0,C 180,E1 -2702.142,E2 -2702.142} C_VEL
LIN {X 0,Y 20.815,Z 773.536,A -85,B 0,C 180,E1 -2716.123,E2 -2716.123} C_VEL
LIN {X 0,Y 8.589,Z 774.114,A -85,B 0,C 180,E1 -2769.559,E2 -2769.559} C_VEL
LIN {X 0,Y 9.83,Z 774.061,A -85,B 0,C 180,E1 -2827.609,E2 -2827.609} C_VEL
LIN {X 0,Y 23.582,Z 773.37,A -85,B 0,C 180,E1 -2867.204,E2 -2867.204} C_VEL
LIN {X 0,Y 41.407,Z 771.652,A -85,B 0,C 180,E1 -2877.895,E2 -2877.895} C_VEL
LIN {X 0,Y 20.438,Z 773.917,A -85,B 0,C 180,E1 -2891.929,E2 -2891.929} C_VEL
LIN {X 0,Y 8.316,Z 774.694,A -85,B 0,C 180,E1 -2948.859,E2 -2948.859} C_VEL
LIN {X 0,Y 8.104,Z 774.736,A -85,B 0,C 180,E1 -2979.292,E2 -2979.292} C_VEL
LIN {X 0,Y 19.515,Z 773.977,A -85,B 0,C 180,E1 -3046.768,E2 -3046.768} C_VEL
LIN {X 0,Y 32.076,Z 772.779,A -85,B 0,C 180,E1 -3058.042,E2 -3058.042} C_VEL
LIN {X 0,Y 30.878,Z 772.881,A -85,B 0,C 180,E1 -3059.863,E2 -3059.863} C_VEL
LIN {X 0,Y 24.06,Z 773.437,A -85,B 0,C 180,E1 -3062.194,E2 -3062.194} C_VEL
LIN {X 0,Y 6.545,Z 774.341,A -85,B 0,C 180,E1 -3064.496,E2 -3064.496} C_VEL
LIN {X 0,Y 0.704,Z 774.458,A -85,B 0,C 180,E1 -3059.005,E2 -3059.005} C_VEL
LIN {X 0,Y 1.381,Z 774.444,A -85,B 0,C 180,E1 -3234.6,E2 -3234.6} C_VEL
LIN {X 0,Y 1.405,Z 774.44,A -85,B 0,C 180,E1 -3063.561,E2 -3063.561} C_VEL
LIN {X 0,Y 0.704,Z 774.458,A -85,B 0,C 180,E1 -3059.005,E2 -3059.005} C_VEL
LIN {X 0,Y 1.261,Z 776.458,A -85,B 0,C 180,E1 -2890.597,E2 -2890.597} C_VEL
LIN {X 0,Y 1.261,Z 799,A -85,B 0,C 180,E1 -2890.597,E2 -2890.597} C_VEL
LIN {X 0,Y 1.261,Z 799,A -85,B 0,C 180,E1 -2890.597,E2 -2890.597}

QRS_NEXT_CUT()

QRS_NEXT()
QRS_HOME()

END
